# EPICS substitutions: viocs/si_ps/si_psApp/Db/cv.substitutions
file "db/individual.db" {
    pattern { family, pos }
        { "CV", "01C1" }
        { "CV", "01C2-A" }
        { "CV", "01C2-B" }
        { "CV", "01C3-A" }
        { "CV", "01C3-B" }
        { "CV", "01C4" }
        { "CV", "01M1" }
        { "CV", "01M2" }
        { "CV", "02C1" }
        { "CV", "02C2-A" }
        { "CV", "02C2-B" }
        { "CV", "02C3-A" }
        { "CV", "02C3-B" }
        { "CV", "02C4" }
        { "CV", "02M1" }
        { "CV", "02M2" }
        { "CV", "03C1" }
        { "CV", "03C2-A" }
        { "CV", "03C2-B" }
        { "CV", "03C3-A" }
        { "CV", "03C3-B" }
        { "CV", "03C4" }
        { "CV", "03M1" }
        { "CV", "03M2" }
        { "CV", "04C1" }
        { "CV", "04C2-A" }
        { "CV", "04C2-B" }
        { "CV", "04C3-A" }
        { "CV", "04C3-B" }
        { "CV", "04C4" }
        { "CV", "04M1" }
        { "CV", "04M2" }
        { "CV", "05C1" }
        { "CV", "05C2-A" }
        { "CV", "05C2-B" }
        { "CV", "05C3-A" }
        { "CV", "05C3-B" }
        { "CV", "05C4" }
        { "CV", "05M1" }
        { "CV", "05M2" }
        { "CV", "06C1" }
        { "CV", "06C2-A" }
        { "CV", "06C2-B" }
        { "CV", "06C3-A" }
        { "CV", "06C3-B" }
        { "CV", "06C4" }
        { "CV", "06M1" }
        { "CV", "06M2" }
        { "CV", "07C1" }
        { "CV", "07C2-A" }
        { "CV", "07C2-B" }
        { "CV", "07C3-A" }
        { "CV", "07C3-B" }
        { "CV", "07C4" }
        { "CV", "07M1" }
        { "CV", "07M2" }
        { "CV", "08C1" }
        { "CV", "08C2-A" }
        { "CV", "08C2-B" }
        { "CV", "08C3-A" }
        { "CV", "08C3-B" }
        { "CV", "08C4" }
        { "CV", "08M1" }
        { "CV", "08M2" }
        { "CV", "09C1" }
        { "CV", "09C2-A" }
        { "CV", "09C2-B" }
        { "CV", "09C3-A" }
        { "CV", "09C3-B" }
        { "CV", "09C4" }
        { "CV", "09M1" }
        { "CV", "09M2" }
        { "CV", "10C1" }
        { "CV", "10C2-A" }
        { "CV", "10C2-B" }
        { "CV", "10C3-A" }
        { "CV", "10C3-B" }
        { "CV", "10C4" }
        { "CV", "10M1" }
        { "CV", "10M2" }
        { "CV", "11C1" }
        { "CV", "11C2-A" }
        { "CV", "11C2-B" }
        { "CV", "11C3-A" }
        { "CV", "11C3-B" }
        { "CV", "11C4" }
        { "CV", "11M1" }
        { "CV", "11M2" }
        { "CV", "12C1" }
        { "CV", "12C2-A" }
        { "CV", "12C2-B" }
        { "CV", "12C3-A" }
        { "CV", "12C3-B" }
        { "CV", "12C4" }
        { "CV", "12M1" }
        { "CV", "12M2" }
        { "CV", "13C1" }
        { "CV", "13C2-A" }
        { "CV", "13C2-B" }
        { "CV", "13C3-A" }
        { "CV", "13C3-B" }
        { "CV", "13C4" }
        { "CV", "13M1" }
        { "CV", "13M2" }
        { "CV", "14C1" }
        { "CV", "14C2-A" }
        { "CV", "14C2-B" }
        { "CV", "14C3-A" }
        { "CV", "14C3-B" }
        { "CV", "14C4" }
        { "CV", "14M1" }
        { "CV", "14M2" }
        { "CV", "15C1" }
        { "CV", "15C2-A" }
        { "CV", "15C2-B" }
        { "CV", "15C3-A" }
        { "CV", "15C3-B" }
        { "CV", "15C4" }
        { "CV", "15M1" }
        { "CV", "15M2" }
        { "CV", "16C1" }
        { "CV", "16C2-A" }
        { "CV", "16C2-B" }
        { "CV", "16C3-A" }
        { "CV", "16C3-B" }
        { "CV", "16C4" }
        { "CV", "16M1" }
        { "CV", "16M2" }
        { "CV", "17C1" }
        { "CV", "17C2-A" }
        { "CV", "17C2-B" }
        { "CV", "17C3-A" }
        { "CV", "17C3-B" }
        { "CV", "17C4" }
        { "CV", "17M1" }
        { "CV", "17M2" }
        { "CV", "18C1" }
        { "CV", "18C2-A" }
        { "CV", "18C2-B" }
        { "CV", "18C3-A" }
        { "CV", "18C3-B" }
        { "CV", "18C4" }
        { "CV", "18M1" }
        { "CV", "18M2" }
        { "CV", "19C1" }
        { "CV", "19C2-A" }
        { "CV", "19C2-B" }
        { "CV", "19C3-A" }
        { "CV", "19C3-B" }
        { "CV", "19C4" }
        { "CV", "19M1" }
        { "CV", "19M2" }
        { "CV", "20C1" }
        { "CV", "20C2-A" }
        { "CV", "20C2-B" }
        { "CV", "20C3-A" }
        { "CV", "20C3-B" }
        { "CV", "20C4" }
        { "CV", "20M1" }
        { "CV", "20M2" }
}
